Omron CX-Programmer project NewProject (CX-Programmer 9.73)

# PLC NewPLC1: CP1E E20

## Global symbols (name address type ; comment)
0.00 BOOL  ; NO1
0.03 BOOL  ; NO3
1.00 BOOL  ; A1
1.01 BOOL  ; NO2
2.00 BOOL  ; A2
2.02 BOOL  ; NC1

## Program NewProgram1 (cyclic task 0)
; LAMPU

### Section Section1

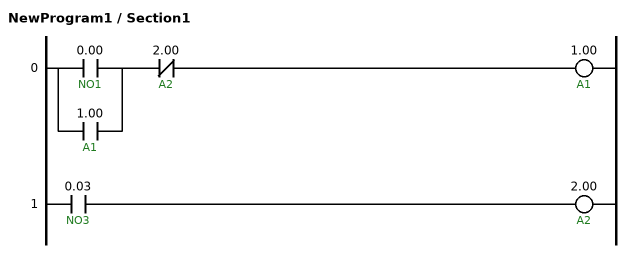
; rung 0
LD 0.00  ; NO1
OR 1.00  ; A1
ANDNOT 2.00  ; A2
OUT 1.00  ; A1
; rung 1
LD 0.03  ; NO3
OUT 2.00  ; A2

### Section END
; rung 0
END(001)